// TIA Portal V18 export
// export: Created 2025-12-01T12:38:06.2978541Z, ExportSetting None, DisplayName Totally Integrated Automation Portal, DisplayVersion V18 Update 5, DisplayName TIA Portal Openness, DisplayVersion V18 Update 5, DisplayName TIA Portal Teamcenter Gateway, DisplayVersion V18, DisplayName TIA Portal Version Control Interface, DisplayVersion V18, DisplayName STEP 7 Professional, DisplayVersion V18 Update 5, DisplayName STEP 7 Safety, DisplayVersion V18, DisplayName WinCC Professional, DisplayVersion V18 Update 5
DATA_BLOCK "ST10_FB_Tower_4Lamp_DB"   // DB5050
// stored: AutoNumber false, InstanceOfName FB_Tower_4Lamp, InstanceOfType FB
"FB_Tower_4Lamp"
   // VAR_INPUT
   //    iReady : Bool;
   //    iManual_Mode : Bool;
   //    iAuto_Mode : Bool;
   //    iAuto_Running : Bool;
   //    iCheck_Mode : Bool;
   //    iIdle : Bool;
   //    iWarning : Bool;
   //    iFault : Bool;
   //    "i0.5s_Pulse" : Bool;
   //    i1s_Pulse : Bool;
   //    i2s_Pulse : Bool;
   //    iResetButton : Bool;
   //    "iE-StopButtonOK" : Bool;
   //    iSafetyGateClosed : Bool;
   //    iSafetyGateRelayOK : Bool;
   //    iPowerOn : Bool;
   //    iMachineHomePos : Bool;
   //    iWorkAreaLightButton : Bool;
   //    iTest_Lamp : Bool;
   // END_VAR
   // VAR_OUTPUT
   //    oRed_Lamp : Bool;
   //    oYellow_Lamp : Bool;
   //    oGreen_Lamp : Bool;
   //    oBlue_Lamp : Bool;
   //    oBuzzer : Bool;
   //    oPowerOn : Bool;
   //    oResetLamp : Bool;
   //    oWorkArea1_LightingOn : Bool;
   //    oWorkArea2_LightingOn : Bool;
   //    oWorkArea3_LightingOn : Bool;
   // END_VAR
   // VAR_IN_OUT
   //    ioStationWaitingLoadPart : Bool;
   //    ioBuzzerON : Bool;
   //    ioBuzzerSetVal : Int;
   // END_VAR
   // VAR
   //    TON : Array[0..10] of TON_TIME;
   //    sRed_Lamp { S7_SetPoint := 'True'} : Bool;
   //    sResetButtonPressed : Bool;
   //    sBuzzerOnCurrentVal : Int;
   //    P_TRIG : Array[0..10] of Bool;
   //    N_TRIG : Array[0..10] of Bool;
   // END_VAR
BEGIN
END_DATA_BLOCK
